// SIMATIC S7-200 project (STEP 7-Micro/WIN), CPU 224XP REL 02.01

SYMBOL_TABLE USER1
sen1             I0.0
sen2             I0.1
sen3             I0.2
sen4             I0.3
sen5             I0.4
sen6             I0.5
sen7             I0.6
c1s1             I0.7
c1s2             I1.0
c2s1             I1.1
c2s2             I1.2
suction          Q0.5
rodless          Q0.3
cyl1             Q0.6
tn1              Q0.4
gripp            Q1.0
cyl2             Q0.1
tn2              Q1.1
con1             Q0.2
con2             Q0.0
con3             Q0.7
END_SYMBOL_TABLE

ORGANIZATION_BLOCK MAIN:OB1
TITLE=PROGRAM COMMENTS
BEGIN
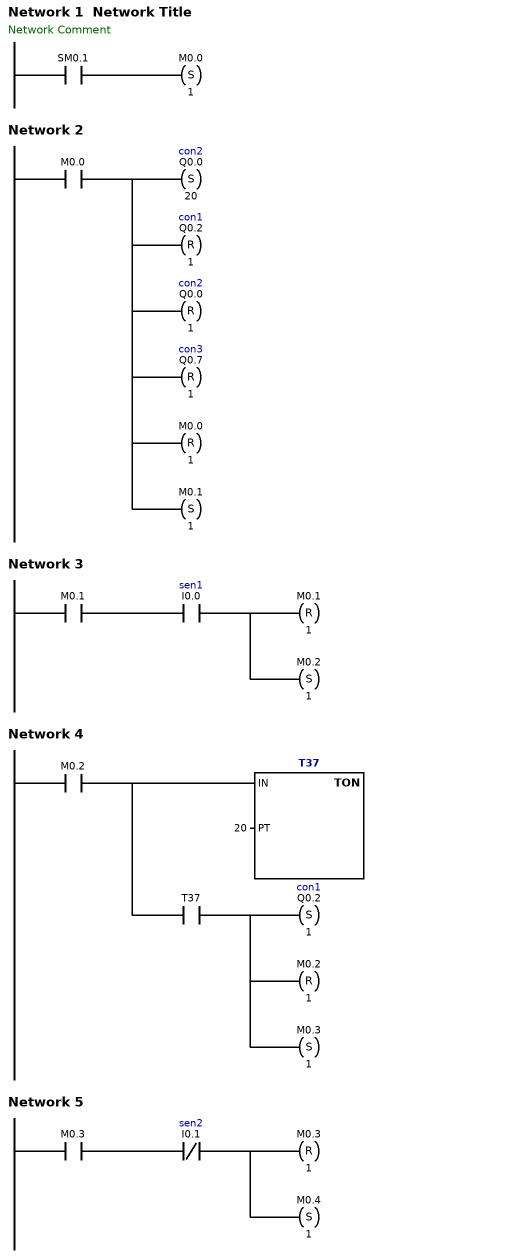
Network 1 // Network Title
// Network Comment
LD     SM0.1
S      M0.0, 1
Network 2
LD     M0.0
S      con2:Q0.0, 20
R      con1:Q0.2, 1
R      con2:Q0.0, 1
R      con3:Q0.7, 1
R      M0.0, 1
S      M0.1, 1
Network 3
LD     M0.1
A      sen1:I0.0
R      M0.1, 1
S      M0.2, 1
Network 4
LD     M0.2
TON    T37, 20
A      T37
S      con1:Q0.2, 1
R      M0.2, 1
S      M0.3, 1
Network 5
LD     M0.3
AN     sen2:I0.1
R      M0.3, 1
S      M0.4, 1
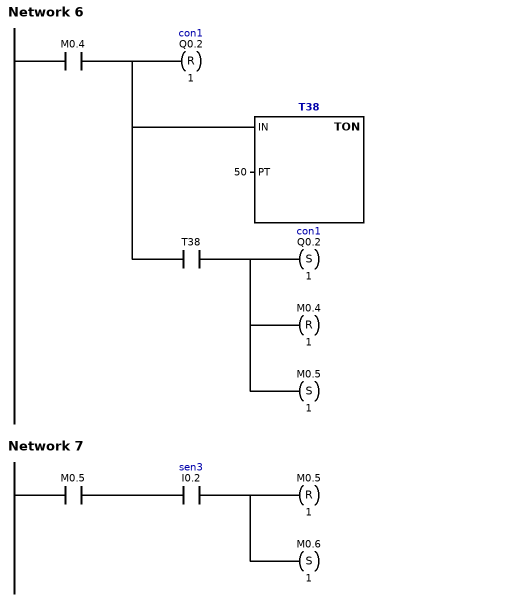
Network 6
LD     M0.4
R      con1:Q0.2, 1
TON    T38, 50
A      T38
S      con1:Q0.2, 1
R      M0.4, 1
S      M0.5, 1
Network 7
LD     M0.5
A      sen3:I0.2
R      M0.5, 1
S      M0.6, 1
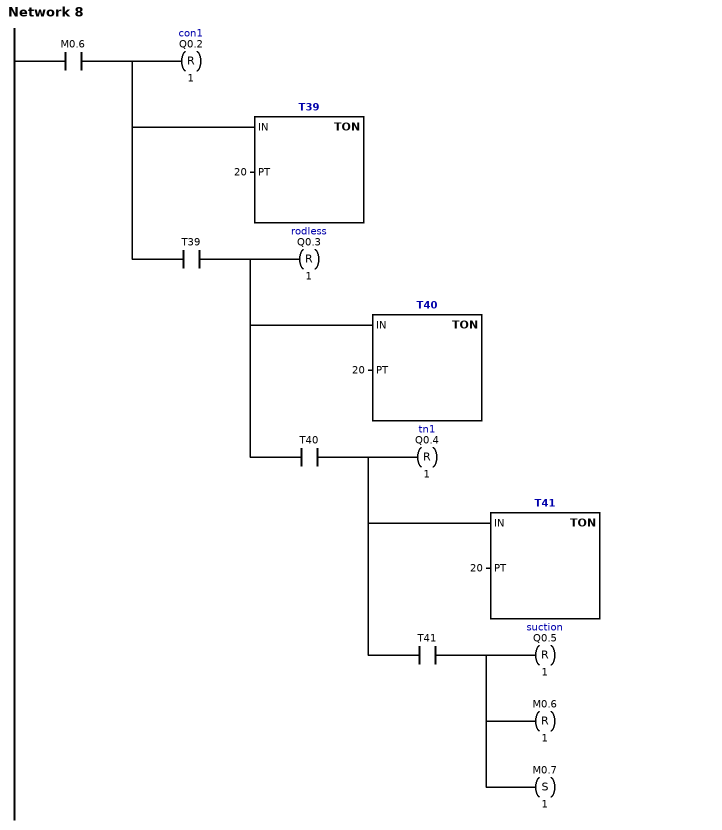
Network 8
LD     M0.6
R      con1:Q0.2, 1
TON    T39, 20
A      T39
R      rodless:Q0.3, 1
TON    T40, 20
A      T40
R      tn1:Q0.4, 1
TON    T41, 20
A      T41
R      suction:Q0.5, 1
R      M0.6, 1
S      M0.7, 1
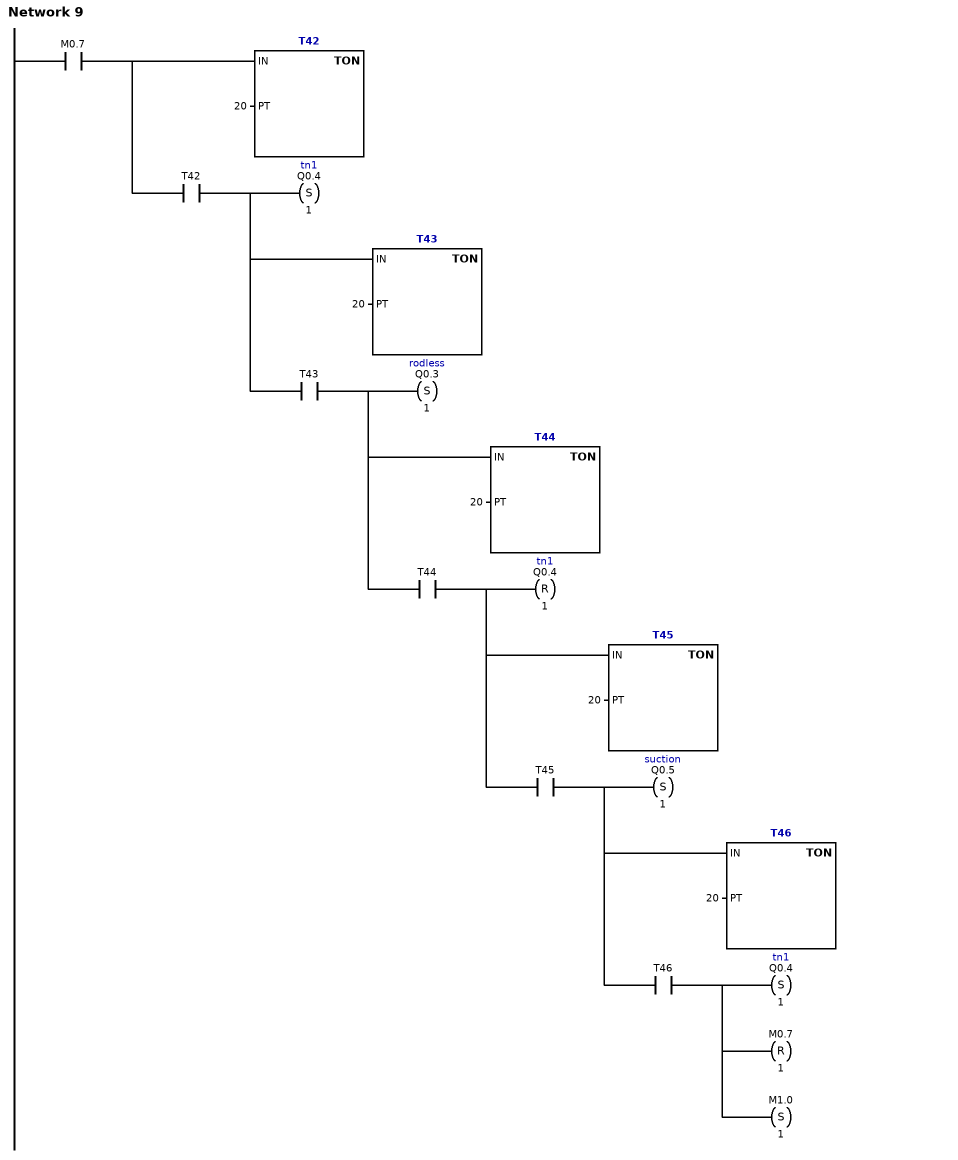
Network 9
LD     M0.7
TON    T42, 20
A      T42
S      tn1:Q0.4, 1
TON    T43, 20
A      T43
S      rodless:Q0.3, 1
TON    T44, 20
A      T44
R      tn1:Q0.4, 1
TON    T45, 20
A      T45
S      suction:Q0.5, 1
TON    T46, 20
A      T46
S      tn1:Q0.4, 1
R      M0.7, 1
S      M1.0, 1
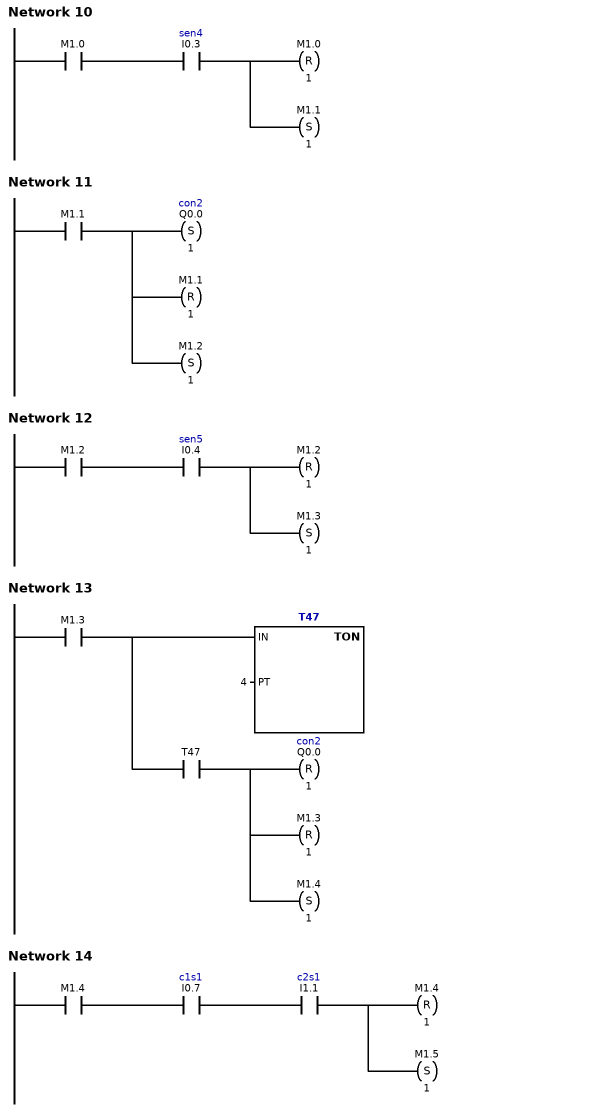
Network 10
LD     M1.0
A      sen4:I0.3
R      M1.0, 1
S      M1.1, 1
Network 11
LD     M1.1
S      con2:Q0.0, 1
R      M1.1, 1
S      M1.2, 1
Network 12
LD     M1.2
A      sen5:I0.4
R      M1.2, 1
S      M1.3, 1
Network 13
LD     M1.3
TON    T47, 4
A      T47
R      con2:Q0.0, 1
R      M1.3, 1
S      M1.4, 1
Network 14
LD     M1.4
A      c1s1:I0.7
A      c2s1:I1.1
R      M1.4, 1
S      M1.5, 1
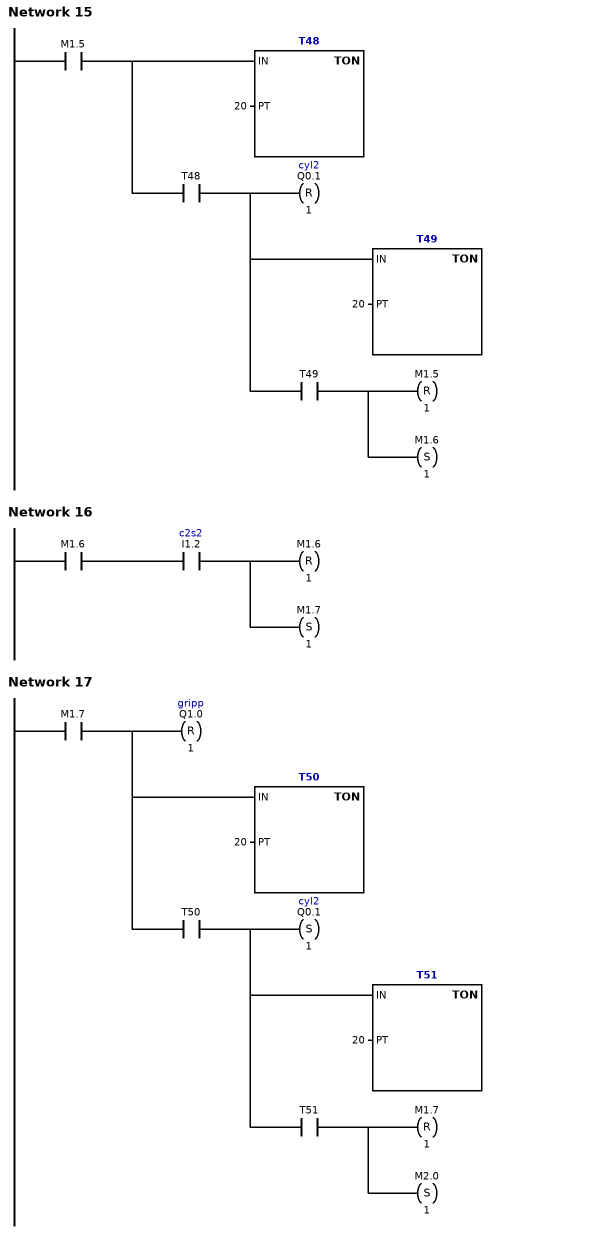
Network 15
LD     M1.5
TON    T48, 20
A      T48
R      cyl2:Q0.1, 1
TON    T49, 20
A      T49
R      M1.5, 1
S      M1.6, 1
Network 16
LD     M1.6
A      c2s2:I1.2
R      M1.6, 1
S      M1.7, 1
Network 17
LD     M1.7
R      gripp:Q1.0, 1
TON    T50, 20
A      T50
S      cyl2:Q0.1, 1
TON    T51, 20
A      T51
R      M1.7, 1
S      M2.0, 1
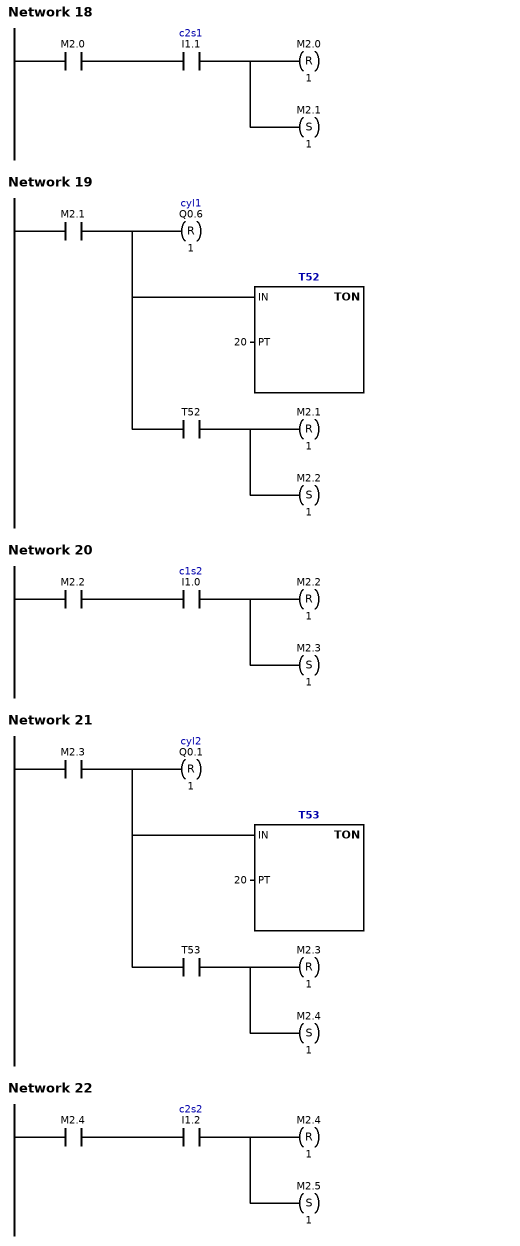
Network 18
LD     M2.0
A      c2s1:I1.1
R      M2.0, 1
S      M2.1, 1
Network 19
LD     M2.1
R      cyl1:Q0.6, 1
TON    T52, 20
A      T52
R      M2.1, 1
S      M2.2, 1
Network 20
LD     M2.2
A      c1s2:I1.0
R      M2.2, 1
S      M2.3, 1
Network 21
LD     M2.3
R      cyl2:Q0.1, 1
TON    T53, 20
A      T53
R      M2.3, 1
S      M2.4, 1
Network 22
LD     M2.4
A      c2s2:I1.2
R      M2.4, 1
S      M2.5, 1
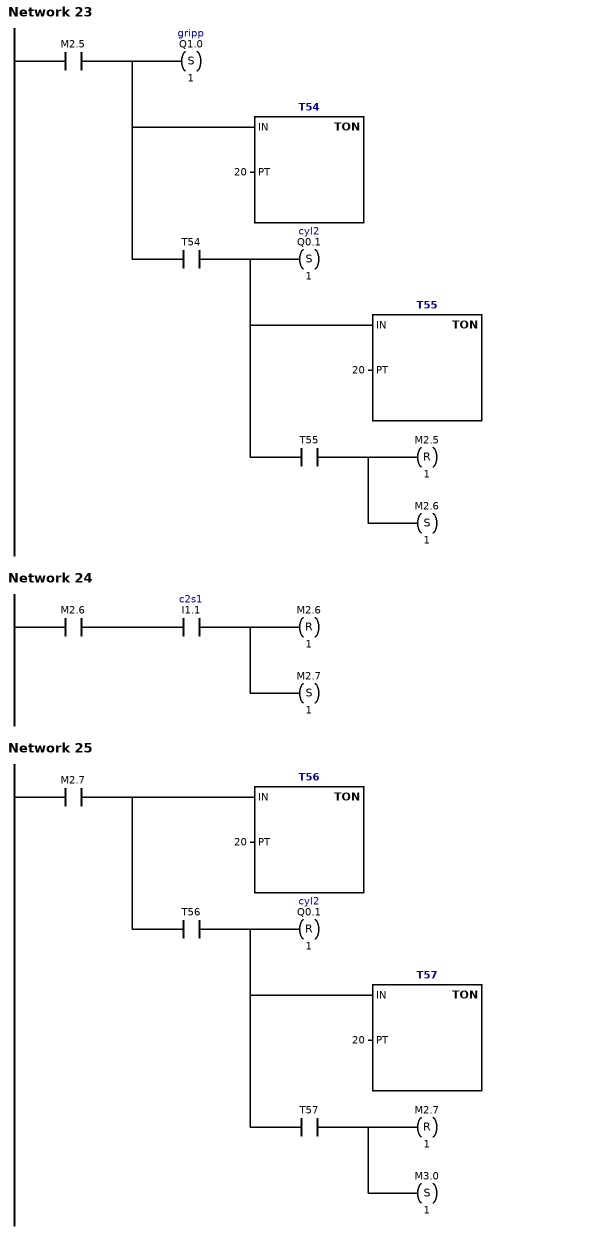
Network 23
LD     M2.5
S      gripp:Q1.0, 1
TON    T54, 20
A      T54
S      cyl2:Q0.1, 1
TON    T55, 20
A      T55
R      M2.5, 1
S      M2.6, 1
Network 24
LD     M2.6
A      c2s1:I1.1
R      M2.6, 1
S      M2.7, 1
Network 25
LD     M2.7
TON    T56, 20
A      T56
R      cyl2:Q0.1, 1
TON    T57, 20
A      T57
R      M2.7, 1
S      M3.0, 1
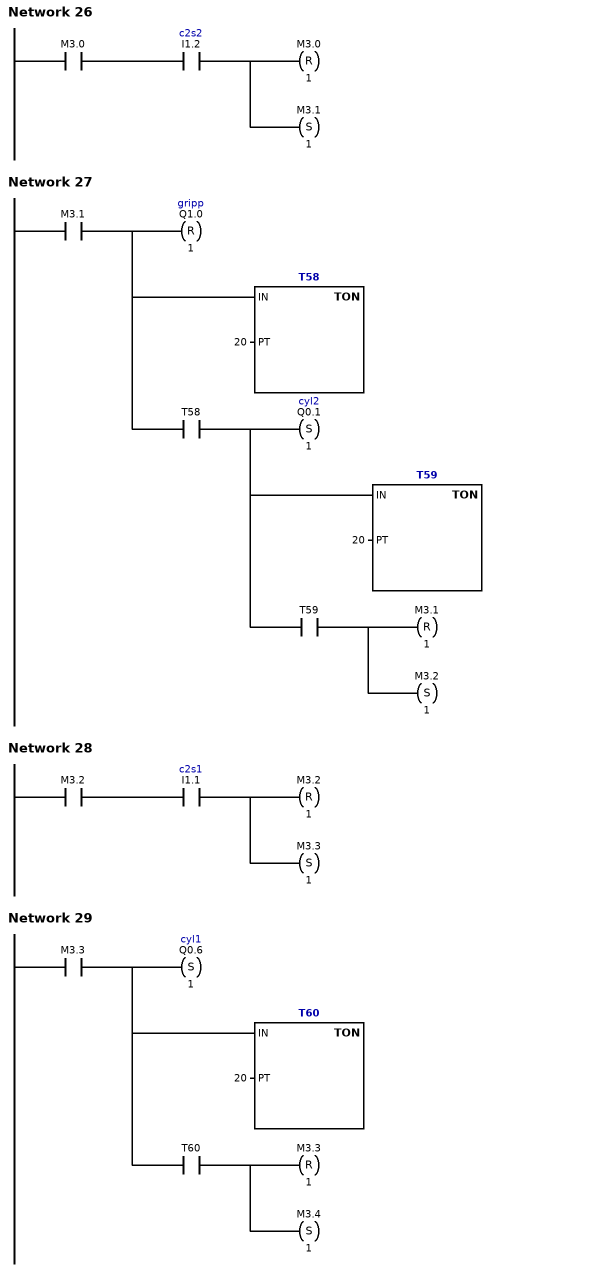
Network 26
LD     M3.0
A      c2s2:I1.2
R      M3.0, 1
S      M3.1, 1
Network 27
LD     M3.1
R      gripp:Q1.0, 1
TON    T58, 20
A      T58
S      cyl2:Q0.1, 1
TON    T59, 20
A      T59
R      M3.1, 1
S      M3.2, 1
Network 28
LD     M3.2
A      c2s1:I1.1
R      M3.2, 1
S      M3.3, 1
Network 29
LD     M3.3
S      cyl1:Q0.6, 1
TON    T60, 20
A      T60
R      M3.3, 1
S      M3.4, 1
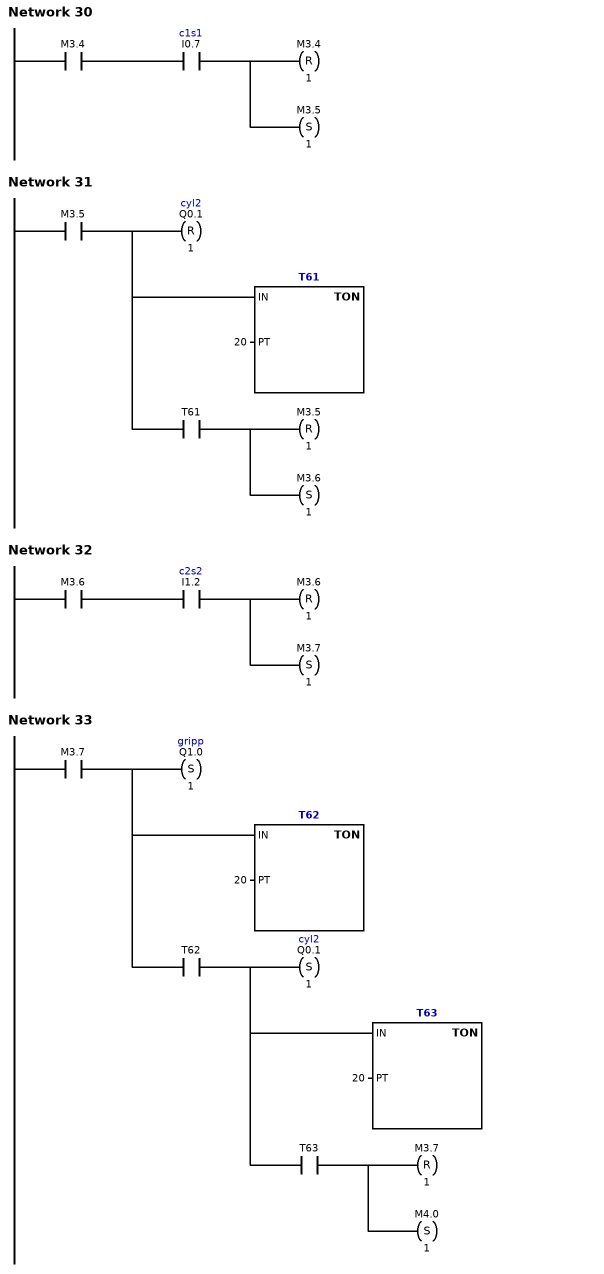
Network 30
LD     M3.4
A      c1s1:I0.7
R      M3.4, 1
S      M3.5, 1
Network 31
LD     M3.5
R      cyl2:Q0.1, 1
TON    T61, 20
A      T61
R      M3.5, 1
S      M3.6, 1
Network 32
LD     M3.6
A      c2s2:I1.2
R      M3.6, 1
S      M3.7, 1
Network 33
LD     M3.7
S      gripp:Q1.0, 1
TON    T62, 20
A      T62
S      cyl2:Q0.1, 1
TON    T63, 20
A      T63
R      M3.7, 1
S      M4.0, 1
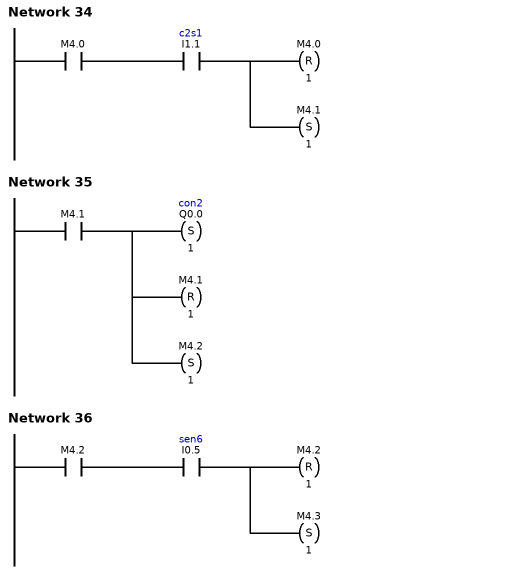
Network 34
LD     M4.0
A      c2s1:I1.1
R      M4.0, 1
S      M4.1, 1
Network 35
LD     M4.1
S      con2:Q0.0, 1
R      M4.1, 1
S      M4.2, 1
Network 36
LD     M4.2
A      sen6:I0.5
R      M4.2, 1
S      M4.3, 1
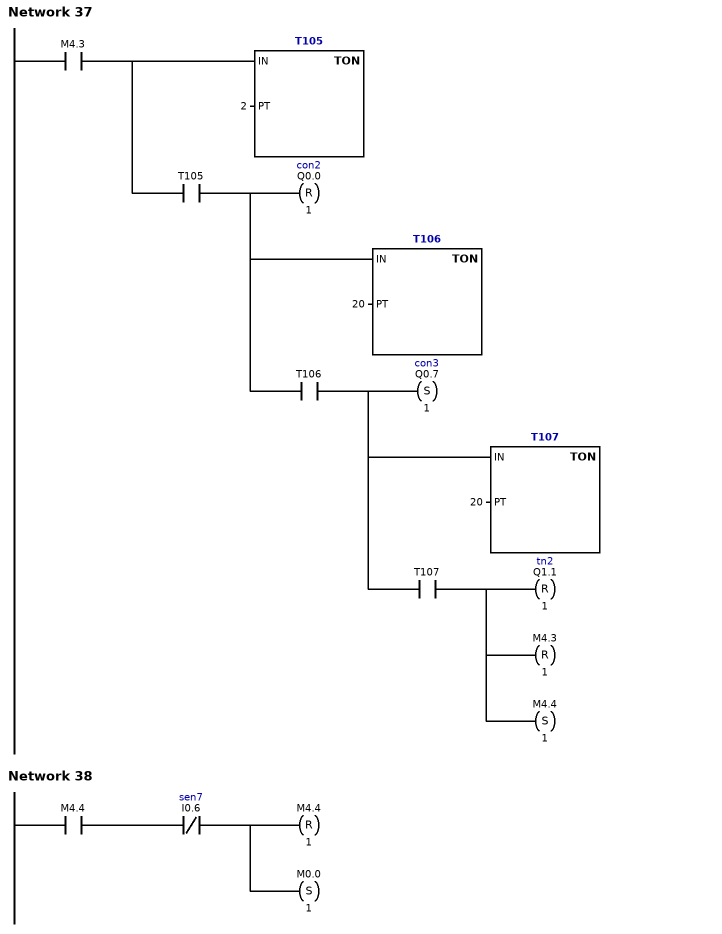
Network 37
LD     M4.3
TON    T105, 2
A      T105
R      con2:Q0.0, 1
TON    T106, 20
A      T106
S      con3:Q0.7, 1
TON    T107, 20
A      T107
R      tn2:Q1.1, 1
R      M4.3, 1
S      M4.4, 1
Network 38
LD     M4.4
AN     sen7:I0.6
R      M4.4, 1
S      M0.0, 1
END_ORGANIZATION_BLOCK
